FUNCTION_BLOCK FB_SteelFurnace EXTENDS FB_StoneFurnace

tProductionTime := T#1.6S;
SUPER^();

{error 'Add property implementation or delete property to use base implementation'}
PROPERTY ProductsOut : UINT
GET
END_GET
END_PROPERTY

END_FUNCTION_BLOCK

(* stored: Version 1.1.0.1, ProductVersion 3.1.4024.13
   POU FB_SteelFurnace: Id {ef0b8919-7282-4bed-bf91-0ac177b2cb7b}, SpecialFunc None
   Property ProductsOut: Id {0e2364c7-469b-47d1-b20f-71e6c2bc9865}
   Get Get: Id {e5a839ce-ed02-4083-bec7-ff54c22f625e} *)
